FUNCTION_BLOCK SKILL_Release (* Names the holder that gives up the equipment a module level skill holds after a failure or abort, for the equipment's release channels (all outputs off, free again) *)
  (* Standard: 61499-2 *)
  (* Version 0.1, 2026-09-28, Project contributors, AAU Smart Production Lab *)
  PACKAGE modlib;
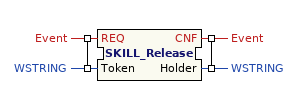
  EVENT_INPUT
    REQ WITH Token;
  END_EVENT
  EVENT_OUTPUT
    CNF WITH Holder;
  END_EVENT
  VAR_INPUT
    Token : WSTRING;
  END_VAR
  VAR_OUTPUT
    Holder : WSTRING;
  END_VAR
  EC_STATES
    REQ : REQ -> CNF;
  END_STATES
  ALGORITHM REQ IN ST:
Holder := Token;
  END_ALGORITHM
END_FUNCTION_BLOCK
